Staubli VAL3: libDialogs.dtx

string VERSION = "0.3.1"
